// TIA Portal V18 export
FUNCTION_BLOCK "laser_centering_device"   // FB4, FBD
{ S7_Optimized_Access := 'TRUE' }
VERSION : 0.1
// stored: AutoNumber true, IsIECCheckEnabled false, IsRetainMemResEnabled false, MemoryReserve 100, SetENOAutomatically false, UDAEnableTagReadback false
   VAR_INPUT
      xBtn : Bool;
      pt_sec : Real;
   END_VAR
   VAR_OUTPUT
      yEnergize : Bool;
   END_VAR
   VAR RETAIN
      pt : Time := T#10s;
   END_VAR
   VAR
      mem : Bool;
      clkBtn : Bool;
      IEC_Timer_0_Instance { S7_SetPoint := 'True'} : TON_TIME;
      xBtnWAS : Bool;
      should_energize_was : Bool;
   END_VAR
BEGIN

REGION Network 2 (SCL)
   #pt := REAL_TO_DINT(#pt_sec * 1000);


   IF #xBtn AND NOT #xBtnWAS THEN
       IF #yEnergize THEN
           #yEnergize := false;
       ELSE
           #yEnergize := TRUE;
       END_IF;
   END_IF;
   #xBtnWAS := #xBtn;
END_REGION

REGION Network 3
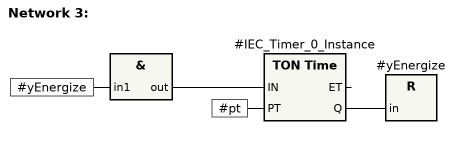
   #IEC_Timer_0_Instance(IN := #yEnergize, PT := #pt);   // TON
   IF #IEC_Timer_0_Instance.Q THEN #yEnergize := FALSE; END_IF;
END_REGION
END_FUNCTION_BLOCK
